{attribute 'linkalways'} 
{attribute 'no_explicit_call' := 'This FB is a CLASS and must be accessed using methods or properties'}
{attribute 'enable_dynamic_creation'}
FUNCTION_BLOCK Node_ContainerType_Vector_TcVnPoint2_LREAL EXTENDS Node
VAR
    out : _GUID;
END_VAR

METHOD PUBLIC  Clone : I_Node
VAR
	pNode : POINTER TO Node_ContainerType_Vector_TcVnPoint2_LREAL;
END_VAR
pNode := __NEW(Node_ContainerType_Vector_TcVnPoint2_LREAL);
Clone := pNode^;
END_METHOD

METHOD FB_init : BOOL
VAR_INPUT
	bInitRetains : BOOL; // if TRUE, the retain variables are initialized (warm start / cold start)
	bInCopyCode : BOOL;  // if TRUE, the instance afterwards gets moved into the copy code (online change)
END_VAR
AddOutput('out', out);
END_METHOD

METHOD PROTECTED OnExecute
out.Value := ContainerType_Vector_TcVnPoint2_LREAL;
END_METHOD

END_FUNCTION_BLOCK

(* stored: Version 1.1.0.1, ProductVersion 3.1.4026.17
   POU Node_ContainerType_Vector_TcVnPoint2_LREAL: Id {e6b50220-c5cd-0a77-03a4-40d0ad5b85d3}, SpecialFunc None
   Folder Constructor: Id {e94997b2-40b9-01e0-080d-ba066bd0995f}
   Method Clone: Id {d4f03bec-af5a-077e-2c32-3e08c9f60eef}
   Method FB_init: Id {5bc70fe9-c4d3-0b92-2a3b-ad63fe559894}
   Method OnExecute: Id {6ff9c872-1c9d-086c-3c6c-b8ce55ea2536} *)
